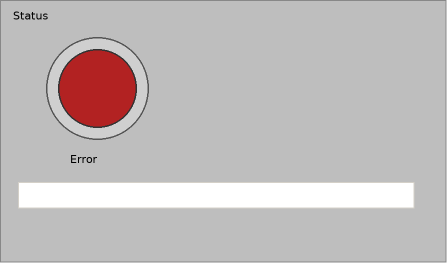
VISUALIZATION Visu2_StatusSimple  // 447x263
    Rectangle (-2,-2 447x263)
    Lamp1 (29,29 137x119), variable: fbBtn.xAru=0 OR stParam.stStatus.xErreur, style: Lamp-Lamp1-Red
    Textfield (18,182 396x26), text variable: stParam.stStatus.sMessage, text list: 'ErrorList', text index: stParam.stStatus.iId
    Label (10,1 176x30), "Status"
    Label (56,145 55x29), "Error"
END_VISUALIZATION

(* stored: Version 1.1.0.1, ProductVersion 3.1.4020.12
   Visu Visu2_StatusSimple: Id {fb344a76-4fbc-4fb6-87de-c054627ed418} *)
